NETWORK
TITLE =SK_A5_START_Molch_L  Anlage 5 Lampe Start Molch IM SIRUPRAUM
// Act 009
// Box           : AB-SK
// Output address: Q181.5
      CALL FC    70 (
           UnitNo                   := #UnitNo,
           ActRec                   := DB5050.SK_A5_START_Molch_L,
           Typ                      := 0,
           FBa                      := #xTmp,
           FBa2                     := #xTmp,
           Out                      := Q    181.5);

NETWORK
TITLE =SK_A5_MOLCH_BEI_A5_L  Anlage 5 Lampe Molch an A5 IM SIRUPRAUM
// Act 010
// Box           : AB-SK
// Output address: Q181.2
      CALL FC    70 (
           UnitNo                   := #UnitNo,
           ActRec                   := DB5050.SK_A5_MOLCH_BEI_A5_L,
           Typ                      := 0,
           FBa                      := #xTmp,
           FBa2                     := #xTmp,
           Out                      := Q    181.2);

NETWORK
TITLE =SK_A5_MOLCH_IN_SK_L  Anlage 5 Lampe Molch im SK IM SIRUPRAUM
// Act 011
// Box           : AB-SK
// Output address: Q181.3
      CALL FC    70 (
           UnitNo                   := #UnitNo,
           ActRec                   := DB5050.SK_A5_MOLCH_IN_SK_L,
           Typ                      := 0,
           FBa                      := #xTmp,
           FBa2                     := #xTmp,
           Out                      := Q    181.3);

NETWORK
TITLE =EA5_V1  MOLCH A5 V1
// Act 012
// Box           : VSA5
// Input address : I192.4
// Output address: Q192.4
      CALL FC    70 (
           UnitNo                   := #UnitNo,
           ActRec                   := DB5050.EA5_V1,
           Typ                      := 1,
           FBa                      := #xTmp,
           FBa2                     := I    192.4,
           Out                      := Q    192.4);

NETWORK
TITLE =EA5_V2  MOLCH A5 V2
// Act 013
// Box           : VSA5
// Input address : I192.5
// Output address: Q192.5
      CALL FC    70 (
           UnitNo                   := #UnitNo,
           ActRec                   := DB5050.EA5_V2,
           Typ                      := 1,
           FBa                      := #xTmp,
           FBa2                     := I    192.5,
           Out                      := Q    192.5);

NETWORK
TITLE =EA5_V31  MOLCH A5 V31 ohne RM
// Act 014
// Box           : VSA5
// Output address: Q192.0
      CALL FC    70 (
           UnitNo                   := #UnitNo,
           ActRec                   := DB5050.EA5_V31,
           Typ                      := 0,
           FBa                      := #xTmp,
           FBa2                     := #xTmp,
           Out                      := Q    192.0);

NETWORK
TITLE =EA5_V32  MOLCH A5 V31 ohne RM
// Act 015
// Box           : VSA5
// Input address : I192.1
// Output address: Q192.1
      CALL FC    70 (
           UnitNo                   := #UnitNo,
           ActRec                   := DB5050.EA5_V32,
           Typ                      := 0,
           FBa                      := #xTmp,
           FBa2                     := I    192.1,
           Out                      := Q    192.1);

NETWORK
TITLE =EA5_V41  MOLCH A5 V41
// Act 016
// Box           : VSA5
// Input address : I192.2
// Output address: Q192.2
      CALL FC    70 (
           UnitNo                   := #UnitNo,
           ActRec                   := DB5050.EA5_V41,
           Typ                      := 1,
           FBa                      := #xTmp,
           FBa2                     := I    192.2,
           Out                      := Q    192.2);

NETWORK
TITLE =EA5_V42  MOLCH A5 V42
// Act 017
// Box           : VSA5
// Input address : I192.3
// Output address: Q192.3
      CALL FC    70 (
           UnitNo                   := #UnitNo,
           ActRec                   := DB5050.EA5_V42,
           Typ                      := 1,
           FBa                      := #xTmp,
           FBa2                     := I    192.3,
           Out                      := Q    192.3);

NETWORK
TITLE =A5_MOLCH_LDT_Start  MOLCH A5 Reserve 23
// Act 019
// Box           : VSA5
// Output address: Q194.7
      CALL FC    70 (
           UnitNo                   := #UnitNo,
           ActRec                   := DB5050.A5_MOLCH_LDT_Start,
           Typ                      := 0,
           FBa                      := #xTmp,
           FBa2                     := #xTmp,
           Out                      := Q    194.7);

NETWORK
TITLE =Molch ist unterwegs(Mixer)


      CALL FC    70 (
           UnitNo                   := #UnitNo,
           ActRec                   := DB5050.Act20,
           Typ                      := 0,
           FBa                      := #xTmp,
           FBa2                     := #xTmp,
           Out                      := Q    199.3);

NETWORK
TITLE =Molch in Endposition (Mixer)


      CALL FC    70 (
           UnitNo                   := #UnitNo,
           ActRec                   := DB5050.Act21,
           Typ                      := 0,
           FBa                      := #xTmp,
           FBa2                     := #xTmp,
           Out                      := Q    199.7);

NETWORK
TITLE =A5_GOA501  Mixer A5 GOA501 Paneel CIP
// Act 025
// Box           : Mixer5
// Output address: Q199.2
      CALL FC    70 (
           UnitNo                   := #UnitNo,
           ActRec                   := DB5050.A5_GOA501,
           Typ                      := 0,
           FBa                      := #xTmp,
           FBa2                     := #xTmp,
           Out                      := Q    199.2);

NETWORK
TITLE =A5_GOA502  Mixer A5 GOA502 Paneel CIP
// Act 027
// Box           : Mixer5
// Output address: Q199.4
      CALL FC    70 (
           UnitNo                   := #UnitNo,
           ActRec                   := DB5050.A5_GOA502,
           Typ                      := 0,
           FBa                      := #xTmp,
           FBa2                     := #xTmp,
           Out                      := Q    199.4);

NETWORK
TITLE =A5_Schwenkbogen  "1"=CIP  "0"=Produktion
// Act 028
// Box           : Sirup
// Output address: DB_SEND_DOEHLER.Anlage5.Schwenkbogen
      CALL FC    70 (
           UnitNo                   := #UnitNo,
           ActRec                   := DB5050.A5_Schwenkbogen,
           Typ                      := 0,
           FBa                      := #xTmp,
           FBa2                     := #xTmp,
           Out                      := DB404.DBX   49.0);

NETWORK
TITLE =A5_GOA503  Mixer A5 GOA503 Paneel CIP
// Act 029
// Box           : Mixer5
// Output address: Q199.5
      CALL FC    70 (
           UnitNo                   := #UnitNo,
           ActRec                   := DB5050.A5_GOA503,
           Typ                      := 0,
           FBa                      := #xTmp,
           FBa2                     := #xTmp,
           Out                      := Q    199.5);

NETWORK
TITLE =VNI_A5_SCHWENKBOGEN_RL  Schwenkbogen A5-RL liegt richtig
// Act 042
// Box           : AB-SK
// Output address: Q183.1
      CALL FC    70 (
           UnitNo                   := #UnitNo,
           ActRec                   := DB5050.VNI_A5_SCHWENKBOGEN_RL,
           Typ                      := 0,
           FBa                      := #xTmp,
           FBa2                     := #xTmp,
           Out                      := Q    183.1);

NETWORK
TITLE =VNI_MOLCH_verr_A5  SIGNAL AN VNI Molch verriegelt an Anlage5
// Act 043
// Box           : AB-SK
// Output address: Q183.2
      CALL FC    70 (
           UnitNo                   := #UnitNo,
           ActRec                   := DB5050.VNI_MOLCH_verr_A5,
           Typ                      := 0,
           FBa                      := #xTmp,
           FBa2                     := #xTmp,
           Out                      := Q    183.2);

NETWORK
TITLE =VNI_MOLCH_Sender_A5  SIGNAL AN VNI Molch an Sendestation A5 (SK)
// Act 044
// Box           : AB-SK
// Output address: Q183.3
      CALL FC    70 (
           UnitNo                   := #UnitNo,
           ActRec                   := DB5050.VNI_MOLCH_Sender_A5,
           Typ                      := 0,
           FBa                      := #xTmp,
           FBa2                     := #xTmp,
           Out                      := Q    183.3);

NETWORK
TITLE =VNI_MOLCH_Empfang_A5  Molch an Empfangsstation (M5)
// Act 045
// Box           : AB-SK
// Output address: Q183.4
      CALL FC    70 (
           UnitNo                   := #UnitNo,
           ActRec                   := DB5050.VNI_MOLCH_Empfang_A5,
           Typ                      := 0,
           FBa                      := #xTmp,
           FBa2                     := #xTmp,
           Out                      := Q    183.4);

NETWORK
TITLE =A5_Molch_Sirup  "1"=Molch ist im Sirupraum
// Act 046
// Box           : Sirup
// Output address: DB_SEND_DOEHLER.Anlage5.Molch_Sirup
      CALL FC    70 (
           UnitNo                   := #UnitNo,
           ActRec                   := DB5050.A5_Molch_Sirup,
           Typ                      := 0,
           FBa                      := #xTmp,
           FBa2                     := #xTmp,
           Out                      := DB404.DBX   48.0);

NETWORK
TITLE =A5_Molch_Anlage  "1"=Molch ist an der Anlage
// Act 047
// Box           : Sirup
// Output address: DB_SEND_DOEHLER.Anlage5.Molch_Anlage
      CALL FC    70 (
           UnitNo                   := #UnitNo,
           ActRec                   := DB5050.A5_Molch_Anlage,
           Typ                      := 0,
           FBa                      := #xTmp,
           FBa2                     := #xTmp,
           Out                      := DB404.DBX   48.1);

NETWORK
TITLE =A5_Molch_PRO  "1"=Molch ist bereit für Produktion
// Act 048
// Box           : Sirup
// Output address: DB_SEND_DOEHLER.Anlage5.Molch_PRO
      CALL FC    70 (
           UnitNo                   := #UnitNo,
           ActRec                   := DB5050.A5_Molch_PRO,
           Typ                      := 0,
           FBa                      := #xTmp,
           FBa2                     := #xTmp,
           Out                      := DB404.DBX   48.2);

NETWORK
TITLE =A5_Molch_CIP  "1"=Molch ist bereit für CIP
// Act 049
// Box           : Sirup
// Output address: DB_SEND_DOEHLER.Anlage5.Molch_CIP
      CALL FC    70 (
           UnitNo                   := #UnitNo,
           ActRec                   := DB5050.A5_Molch_CIP,
           Typ                      := 0,
           FBa                      := #xTmp,
           FBa2                     := #xTmp,
           Out                      := DB404.DBX   48.3);

NETWORK
TITLE =A5_Sirupanforderung
// Act 050
// Box           : Sirup
// Output address: DB_SEND_DOEHLER.Anlage5.Sirupanforderung
      CALL FC    70 (
           UnitNo                   := #UnitNo,
           ActRec                   := DB5050.A5_Sirupanforderung,
           Typ                      := 0,
           FBa                      := #xTmp,
           FBa2                     := #xTmp,
           Out                      := DB404.DBX   48.4);

END_FUNCTION_BLOCK

FUNCTION_BLOCK FB 4051
TITLE =U105: Transfer Plant 5
FAMILY : BOTEC_F1
NAME : UniE
VERSION : 1.2


VAR_TEMP
  CIP : BOOL ;	//CIP active
  UNIM : BOOL ;	//Unit Not In Maintenance
  GenRel : BOOL ;	//general OK (emergency and maintenance OK)
  EStopOK : BOOL ;	//emergency OK
  UnitNo : INT ;	//unit number
  xTmp : BOOL ;	//Temporary Bool
  iTmp : INT ;	//Temporary INT
  rTmp : REAL ;	//Temporary REAL
  dTmp : DINT ;	//Temporary DINT (free for general use)
  RetValInt : INT ;	//return value
END_VAR
BEGIN
NETWORK
TITLE =General

      SET   ;
// Simulation ---------------------------------------------------------------
      A     DB4051.DBX 1357.7;
      CC    FB  4059; // "U105Sim"
      A     DB4051.DBX   17.3;
      =     DB4051.DBX 1357.7; //Help bit for simulation

// get unit number ----------------------------------------------------------
      L     DB4050.DBW    0;
      T     #UnitNo;

// communication ------------------------------------------------------------
      UC    FB  4055; // U105Com

NETWORK
TITLE =Sequence organisation

      CLR   ;
      =     M    122.2;

// sequencer ----------------------------------------------------------------
      A     DB4053.DBX   43.1;
      S     DB4053.DBX   97.3;

      CALL FC    40 (
           UnitNo                   := #UnitNo);

END_FUNCTION_BLOCK

FUNCTION_BLOCK FB 4070
TITLE =U107: Sirup Anlage  7
FAMILY : BOTEC_F1
NAME : U107A
VERSION : 2.1


VAR_TEMP
  EStopOK : BOOL ;	//auxiliary flag
  CIP : BOOL ;	//CIP Program Selected
  xTmp : BOOL ;	//Temporary Bool(free for general use)
  DummyBool : BOOL ;	//Temporary Bool(free for general use)
  UnitNo : INT ;	//unit number
  UnitFB : INT ;	//unit expansion FB number
  rTmp : REAL ;	//Temporary REAL (free for general use)
  iTmp : INT ;	//Temporary INT (free for general use)
  DummyInt : INT ;	//Temporary INT (free for general use)
  dTmp : DINT ;	//Temporary DINT (free for general use)
END_VAR
BEGIN
NETWORK
TITLE =general

      CLR   ;
      =     #xTmp;
      =     #EStopOK;

      L     DB4070.DBW    0;
      T     #UnitNo;
      L     DB4070.DBW    2;
      T     #UnitFB;

NETWORK
TITLE =Universal value

      NOP   0;
// unv001 UnV 001 Process Status
      CALL FC    27 (
           UnitNo                   := #UnitNo,
           UnVRec                   := DB5075.unv001,
           ValExt                   := DB5075.DBD  234);

// unv002 UnV 002 Universal Value 02
      CALL FC    27 (
           UnitNo                   := #UnitNo,
           UnVRec                   := DB5075.unv002,
           ValExt                   := DB5075.DBD  362);

// unv003 UnV 003 Universal Value 03
      CALL FC    27 (
           UnitNo                   := #UnitNo,
           UnVRec                   := DB5075.unv003,
           ValExt                   := DB5075.DBD  490);

// unv004 UnV 004 Universal Value 04
      CALL FC    27 (
           UnitNo                   := #UnitNo,
           UnVRec                   := DB5075.unv004,
           ValExt                   := DB5075.DBD  618);

NETWORK
TITLE =special inputs

      NOP   0;
// GOA_SA7_3_1_oben SpI 004
      CALL FC    14 (
           UnitNo                   := #UnitNo,
           SpIRec                   := DB5071.GOA_SA7_3_1_oben,
           SpIBit                   := I     74.2);

// GOA_SA7_3_2_unten SpI 005 Korb im Sirupraum in unterer Position
      CALL FC    14 (
           UnitNo                   := #UnitNo,
           SpIRec                   := DB5071.GOA_SA7_3_2_unten,
           SpIBit                   := I     74.3);

// GOA_SA7_1 SpI 006
      CALL FC    14 (
           UnitNo                   := #UnitNo,
           SpIRec                   := DB5071.GOA_SA7_1,
           SpIBit                   := I     74.1);// "GOA_SA7_1"

// GOA_SA7_2 SpI 007
      CALL FC    14 (
           UnitNo                   := #UnitNo,
           SpIRec                   := DB5071.GOA_SA7_2,
           SpIBit                   := I     74.0);//"GOA_SA7_2"

// SK_A7_Molch_Abbruch_DT SpI 008 MOLCH A7 Drucktaste Abbruch Sirupraum
      CALL FC    14 (
           UnitNo                   := #UnitNo,
           SpIRec                   := DB5071.SK_A7_Molch_Abbruch_DT,
           SpIBit                   := I    180.0);

// SK_A7_START_Molch_LDT SpI 009 MOLCH A7 L-Drucktaste Start Sirupraum
      CALL FC    14 (
           UnitNo                   := #UnitNo,
           SpIRec                   := DB5071.SK_A7_START_Molch_LDT,
           SpIBit                   := I    180.3);

// A7_Sk1_Handklappe SpI 010
      CALL FC    14 (
           UnitNo                   := #UnitNo,
           SpIRec                   := DB5071.A7_Sk1_Handklappe,
           SpIBit                   := I     74.7);

// GOA_EA7_3_1_oben SpI 014
      CALL FC    14 (
           UnitNo                   := #UnitNo,
           SpIRec                   := DB5071.GOA_EA7_3_1_oben,
           SpIBit                   := I     26.5);

// GOA_EA7_3_2_unten SpI 015
      CALL FC    14 (
           UnitNo                   := #UnitNo,
           SpIRec                   := DB5071.GOA_EA7_3_2_unten,
           SpIBit                   := I     26.6);

// GOA_EA7_3 SpI 016 Molch in Startposition an Anlage 7
      CALL FC    14 (
           UnitNo                   := #UnitNo,
           SpIRec                   := DB5071.GOA_EA7_3,
           SpIBit                   := I     26.3);

// GOA_EA7_4 SpI 017 GOA Molch in Ruhelage an Anlage 7
      CALL FC    14 (
           UnitNo                   := #UnitNo,
           SpIRec                   := DB5071.GOA_EA7_4,
           SpIBit                   := I     26.4);

// A7_SS_FRG_MOLCH SpI 018 Anlage 7 Schlüsselschalter Freigabe Molch
      CALL FC    14 (
           UnitNo                   := #UnitNo,
           SpIRec                   := DB5071.A7_SS_FRG_MOLCH,
           SpIBit                   := I     27.4);

// LDT_START_MOLCH_S2 SpI 019 STARTTASTER AB
      CALL FC    14 (
           UnitNo                   := #UnitNo,
           SpIRec                   := DB5071.LDT_START_MOLCH_S2,
           SpIBit                   := I     26.7);

// LDT_STOP_MOLCH_S2 SpI 020
      CALL FC    14 (
           UnitNo                   := #UnitNo,
           SpIRec                   := DB5071.LDT_STOP_MOLCH_S2,
           SpIBit                   := I     27.5);

// EA7_K2_Handklappe SpI 021 Handklappe Fueller 7
      CALL FC    14 (
           UnitNo                   := #UnitNo,
           SpIRec                   := DB5071.EA7_K2_Handklappe,
           SpIBit                   := I     27.2);

// GOA_701 SpI 022 Spare
      CALL FC    14 (
           UnitNo                   := #UnitNo,
           SpIRec                   := DB5071.GOA_701x,
           SpIBit                   := FALSE);

// GOA_702 SpI 023 Meldung an Fueller/Sirup Anl.7
      CALL FC    14 (
           UnitNo                   := #UnitNo,
           SpIRec                   := DB5071.GOA_702,
           SpIBit                   := I     26.1);

// GOA_701 SpI 025 Meldung an Fueller/Sirup Anl.7
      CALL FC    14 (
           UnitNo                   := #UnitNo,
           SpIRec                   := DB5071.GOA_701,
           SpIBit                   := I     26.0);

NETWORK
TITLE =messages

      NOP   0;
// msg001 Msg 001 Message 01
      CALL FC    16 (
           UnitNo                   := #UnitNo,
           MsgRec                   := DB5077.msg001,
           MsgBit                   := DB5077.DBX   82.7);

// msg002 Msg 002 Message 02
      CALL FC    16 (
           UnitNo                   := #UnitNo,
           MsgRec                   := DB5077.msg002,
           MsgBit                   := DB5077.DBX  142.7);

// msg003 Msg 003 Message 03
      CALL FC    16 (
           UnitNo                   := #UnitNo,
           MsgRec                   := DB5077.msg003,
           MsgBit                   := DB5077.DBX  202.7);

NETWORK
TITLE =unit supply

      UC    FB [#UnitFB];

NETWORK
TITLE =A7_MWV1  Ansteuerung A7_MWV1
// Act 002
// Box           : VSSK
// Input address : I72.4
// Output address: Q52.4
      CALL FC    70 (
           UnitNo                   := #UnitNo,
           ActRec                   := DB5070.A7_MWV1,
           Typ                      := 1,
           FBa                      := #xTmp,
           FBa2                     := I     72.4,
           Out                      := Q     52.4);

NETWORK
TITLE =SA7_V2  Ansteuerung SA7_V2
// Act 003
// Box           : VSSK
// Input address : I72.5
// Output address: Q52.5
      CALL FC    70 (
           UnitNo                   := #UnitNo,
           ActRec                   := DB5070.SA7_V2,
           Typ                      := 3,
           FBa                      := I     72.5,
           FBa2                     := #xTmp,
           Out                      := Q     52.5);

NETWORK
TITLE =SA7_V31  Ansteuerung SA7_V31 ohne RM
// Act 004
// Box           : VSSK
// Output address: Q52.0
      CALL FC    70 (
           UnitNo                   := #UnitNo,
           ActRec                   := DB5070.SA7_V31,
           Typ                      := 0,
           FBa                      := #xTmp,
           FBa2                     := #xTmp,
           Out                      := Q     52.0);

NETWORK
TITLE =SA7_V32  Ansteuerung SA7_V32 ohne RM
// Act 005
// Box           : VSSK
// Output address: Q52.1
      CALL FC    70 (
           UnitNo                   := #UnitNo,
           ActRec                   := DB5070.SA7_V32,
           Typ                      := 0,
           FBa                      := #xTmp,
           FBa2                     := #xTmp,
           Out                      := Q     52.1);

NETWORK
TITLE =SA7_V41  Ansteuerung SA7_V41
// Act 006
// Box           : VSSK
// Input address : I72.2
// Output address: Q52.2
      CALL FC    70 (
           UnitNo                   := #UnitNo,
           ActRec                   := DB5070.SA7_V41,
           Typ                      := 3,
           FBa                      := I     72.2,
           FBa2                     := #xTmp,
           Out                      := Q     52.2);

NETWORK
TITLE =SA7_V42  Ansteuerung SA7_V42
// Act 007
// Box           : VSSK
// Input address : I72.3
// Output address: Q52.3
      CALL FC    70 (
           UnitNo                   := #UnitNo,
           ActRec                   := DB5070.SA7_V42,
           Typ                      := 3,
           FBa                      := I     72.3,
           FBa2                     := #xTmp,
           Out                      := Q     52.3);

NETWORK
TITLE =SK_A7_Abbruch_L  Anlage 7 Lampe Abbruch IM SIRUPRAUM
// Act 008
// Box           : AB-SK
// Output address: Q180.2
      CALL FC    70 (
           UnitNo                   := #UnitNo,
           ActRec                   := DB5070.SK_A7_Abbruch_L,
           Typ                      := 0,
           FBa                      := #xTmp,
           FBa2                     := #xTmp,
           Out                      := Q    180.2);

NETWORK
TITLE =SK_A7_START_Molch_L  Anlage 7 Lampe Start Molch IM SIRUPRAUM
// Act 009
// Box           : AB-SK
// Output address: Q180.3
      CALL FC    70 (
           UnitNo                   := #UnitNo,
           ActRec                   := DB5070.SK_A7_START_Molch_L,
           Typ                      := 0,
           FBa                      := #xTmp,
           FBa2                     := #xTmp,
           Out                      := Q    180.3);

NETWORK
TITLE =SK_A7_MOLCH_BEI_A7_L  Anlage 7 Lampe Molch an A7 IM SIRUPRAUM
// Act 010
// Box           : AB-SK
// Output address: Q180.0
      CALL FC    70 (
           UnitNo                   := #UnitNo,
           ActRec                   := DB5070.SK_A7_MOLCH_BEI_A7_L,
           Typ                      := 0,
           FBa                      := #xTmp,
           FBa2                     := #xTmp,
           Out                      := Q    180.0);

NETWORK
TITLE =SK_A7_MOLCH_IN_SK_L  Anlage 7 Lampe Molch im SK IM SIRUPRAUM
// Act 011
// Box           : AB-SK
// Output address: Q180.1
      CALL FC    70 (
           UnitNo                   := #UnitNo,
           ActRec                   := DB5070.SK_A7_MOLCH_IN_SK_L,
           Typ                      := 0,
           FBa                      := #xTmp,
           FBa2                     := #xTmp,
           Out                      := Q    180.1);

NETWORK
TITLE =EA7_V1  Molch Anlage 7
// Act 012
// Box           : VSA7
// Input address : I24.4
// Output address: Q46.4
      CALL FC    70 (
           UnitNo                   := #UnitNo,
           ActRec                   := DB5070.EA7_V1,
           Typ                      := 3,
           FBa                      := I     24.4,
           FBa2                     := #xTmp,
           Out                      := Q     46.4);

NETWORK
TITLE =EA7_V2  Molch Anlage 7
// Act 013
// Box           : VSA7
// Input address : I24.5
// Output address: Q46.5
      CALL FC    70 (
           UnitNo                   := #UnitNo,
           ActRec                   := DB5070.EA7_V2,
           Typ                      := 3,
           FBa                      := I     24.5,
           FBa2                     := #xTmp,
           Out                      := Q     46.5);

NETWORK
TITLE =EA7_V31  Molch Anlage 7
// Act 014
// Box           : VSA7
// Output address: Q46.0
      CALL FC    70 (
           UnitNo                   := #UnitNo,
           ActRec                   := DB5070.EA7_V31,
           Typ                      := 0,
           FBa                      := #xTmp,
           FBa2                     := #xTmp,
           Out                      := Q     46.0);

NETWORK
TITLE =EA7_V32  Molch Anlage 7
// Act 015
// Box           : VSA7
// Output address: Q46.1
      CALL FC    70 (
           UnitNo                   := #UnitNo,
           ActRec                   := DB5070.EA7_V32,
           Typ                      := 0,
           FBa                      := #xTmp,
           FBa2                     := #xTmp,
           Out                      := Q     46.1);

NETWORK
TITLE =EA7_V41  Molch Anlage 7
// Act 016
// Box           : VSA7
// Input address : I24.2
// Output address: Q46.2
      CALL FC    70 (
           UnitNo                   := #UnitNo,
           ActRec                   := DB5070.EA7_V41,
           Typ                      := 3,
           FBa                      := I     24.2,
           FBa2                     := #xTmp,
           Out                      := Q     46.2);

NETWORK
TITLE =EA7_V42  Molch Anlage 7
// Act 017
// Box           : VSA7
// Input address : I24.3
// Output address: Q46.3
      CALL FC    70 (
           UnitNo                   := #UnitNo,
           ActRec                   := DB5070.EA7_V42,
           Typ                      := 3,
           FBa                      := I     24.3,
           FBa2                     := #xTmp,
           Out                      := Q     46.3);

NETWORK
TITLE =LA_S2_MOLCH_START  LAMPE LDT AB
// Act 019
// Box           : FRM-A7
// Output address: Q59.7
      CALL FC    70 (
           UnitNo                   := #UnitNo,
           ActRec                   := DB5070.LA_S2_MOLCH_START,
           Typ                      := 0,
           FBa                      := #xTmp,
           FBa2                     := #xTmp,
           Out                      := Q     59.7);

NETWORK
TITLE =Molch ist unterwegs (Mixer)


      CALL FC    70 (
           UnitNo                   := #UnitNo,
           ActRec                   := DB5070.Act20,
           Typ                      := 0,
           FBa                      := #xTmp,
           FBa2                     := #xTmp,
           Out                      := Q     59.3);

NETWORK
TITLE =Molch in Endposition (Mixer)


      CALL FC    70 (
           UnitNo                   := #UnitNo,
           ActRec                   := DB5070.Act21,
           Typ                      := 0,
           FBa                      := #xTmp,
           FBa2                     := #xTmp,
           Out                      := Q     59.6);

NETWORK
TITLE =A7_GOA_701  Meldung an Fueller/Sirup Anl.7
// Act 022
// Box           : FRM-A7
// Output address: Q59.2
      CALL FC    70 (
           UnitNo                   := #UnitNo,
           ActRec                   := DB5070.A7_GOA_701,
           Typ                      := 0,
           FBa                      := #xTmp,
           FBa2                     := #xTmp,
           Out                      := Q     59.2);

NETWORK
TITLE =A7_GOA_702  Meldung an Fueller/Mixer Anl.7
// Act 023
// Box           : FRM-A7
// Output address: Q59.5
      CALL FC    70 (
           UnitNo                   := #UnitNo,
           ActRec                   := DB5070.A7_GOA_702,
           Typ                      := 0,
           FBa                      := #xTmp,
           FBa2                     := #xTmp,
           Out                      := Q     59.5);

NETWORK
TITLE =A7_GOA_703  Meldung an Fueller/Mixer Anl.7
// Act 024
// Box           : FRM-A7
// Output address: Q59.4
      CALL FC    70 (
           UnitNo                   := #UnitNo,
           ActRec                   := DB5070.A7_GOA_703,
           Typ                      := 0,
           FBa                      := #xTmp,
           FBa2                     := #xTmp,
           Out                      := Q     59.4);

NETWORK
TITLE =A7_Schwenkbogen  "1"=CIP  "0"=Produktion
// Act 028
// Box           : Sirup
// Output address: DB_SEND_DOEHLER.Anlage7.Schwenkbogen
      CALL FC    70 (
           UnitNo                   := #UnitNo,
           ActRec                   := DB5070.A7_Schwenkbogen,
           Typ                      := 0,
           FBa                      := #xTmp,
           FBa2                     := #xTmp,
           Out                      := DB404.DBX   53.0);

NETWORK
TITLE =A7_Molch_Sirup  "1"=Molch ist im Sirupraum
// Act 046
// Box           : Sirup
// Output address: DB_SEND_DOEHLER.Anlage7.Molch_Sirup
      CALL FC    70 (
           UnitNo                   := #UnitNo,
           ActRec                   := DB5070.A7_Molch_Sirup,
           Typ                      := 0,
           FBa                      := #xTmp,
           FBa2                     := #xTmp,
           Out                      := DB404.DBX   52.0);

NETWORK
TITLE =A7_Molch_Anlage  "1"=Molch ist an der Anlage
// Act 047
// Box           : Sirup
// Output address: DB_SEND_DOEHLER.Anlage7.Molch_Anlage
      CALL FC    70 (
           UnitNo                   := #UnitNo,
           ActRec                   := DB5070.A7_Molch_Anlage,
           Typ                      := 0,
           FBa                      := #xTmp,
           FBa2                     := #xTmp,
           Out                      := DB404.DBX   52.1);

NETWORK
TITLE =A7_Molch_PRO  "1"=Molch ist bereit für Produktion
// Act 048
// Box           : Sirup
// Output address: DB_SEND_DOEHLER.Anlage7.Molch_PRO
      CALL FC    70 (
           UnitNo                   := #UnitNo,
           ActRec                   := DB5070.A7_Molch_PRO,
           Typ                      := 0,
           FBa                      := #xTmp,
           FBa2                     := #xTmp,
           Out                      := DB404.DBX   52.2);

NETWORK
TITLE =A7_Molch_CIP  "1"=Molch ist bereit für CIP
// Act 049
// Box           : Sirup
// Output address: DB_SEND_DOEHLER.Anlage7.Molch_CIP
      CALL FC    70 (
           UnitNo                   := #UnitNo,
           ActRec                   := DB5070.A7_Molch_CIP,
           Typ                      := 0,
           FBa                      := #xTmp,
           FBa2                     := #xTmp,
           Out                      := DB404.DBX   52.3);

NETWORK
TITLE =A7_Sirupanforderung
// Act 050
// Box           : Sirup
// Output address: DB_SEND_DOEHLER.Anlage7.Sirupanforderung
      CALL FC    70 (
           UnitNo                   := #UnitNo,
           ActRec                   := DB5070.A7_Sirupanforderung,
           Typ                      := 0,
           FBa                      := #xTmp,
           FBa2                     := #xTmp,
           Out                      := DB404.DBX   52.4);

END_FUNCTION_BLOCK

FUNCTION_BLOCK FB 4071
TITLE =U107: Transfer Plant 7
FAMILY : BOTEC_F1
NAME : UniE
VERSION : 1.2


VAR_TEMP
  CIP : BOOL ;	//CIP active
  UNIM : BOOL ;	//Unit Not In Maintenance
  GenRel : BOOL ;	//general OK (emergency and maintenance OK)
  EStopOK : BOOL ;	//emergency OK
  UnitNo : INT ;	//unit number
  xTmp : BOOL ;	//Temporary Bool
  iTmp : INT ;	//Temporary INT
  rTmp : REAL ;	//Temporary REAL
  dTmp : DINT ;	//Temporary DINT (free for general use)
  RetValInt : INT ;	//return value
END_VAR
BEGIN
NETWORK
TITLE =General

      SET   ;
// Simulation ---------------------------------------------------------------
      A     DB4071.DBX 1357.7;
      CC    FB  4079; // "U107Sim"
      A     DB4071.DBX   17.3;
      =     DB4071.DBX 1357.7; //Help bit for simulation

// get unit number ----------------------------------------------------------
      L     DB4070.DBW    0;
      T     #UnitNo;

// CIP ----------------------------------------------------------------------
      L     DB4071.DBD   54;
      L     0;
      <D    ;
      =     #CIP;

// emergency OK -------------------------------------------------------------
      A     DB4075.DBX   27.0; //Emergency Stop OK
      =     #EStopOK;

// Write Unit in Maintenance ------------------------------------------------

      AN    DB4071.DBX   69.7;
      =     #UNIM;

// emergency and maintenance OK ---------------------------------------------
      A     #EStopOK;
      A     #UNIM;
      =     #GenRel;

// communication ------------------------------------------------------------
      UC    FB  4075; // U107Com

NETWORK
TITLE =Sequence organisation

      CLR   ;
      =     M    122.2;

// SFM supply ----------------------------------------------------------------

// sequencer ----------------------------------------------------------------
      A     DB4073.DBX   43.1;
      S     DB4073.DBX   97.3;

      CALL FC    40 (
           UnitNo                   := #UnitNo);

END_FUNCTION_BLOCK

FUNCTION_BLOCK FB 4080
TITLE =U108: Sirup Anlage  8
FAMILY : BOTEC_F1
NAME : U108A
VERSION : 2.1


VAR_TEMP
  EStopOK : BOOL ;	//auxiliary flag
  CIP : BOOL ;	//CIP Program Selected
  xTmp : BOOL ;	//Temporary Bool(free for general use)
  DummyBool : BOOL ;	//Temporary Bool(free for general use)
  UnitNo : INT ;	//unit number
  UnitFB : INT ;	//unit expansion FB number
  rTmp : REAL ;	//Temporary REAL (free for general use)
  iTmp : INT ;	//Temporary INT (free for general use)
  DummyInt : INT ;	//Temporary INT (free for general use)
  dTmp : DINT ;	//Temporary DINT (free for general use)
END_VAR
BEGIN
NETWORK
TITLE =general

      CLR   ;
      =     #xTmp;
      =     #EStopOK;

      L     DB4080.DBW    0;
      T     #UnitNo;
      L     DB4080.DBW    2;
      T     #UnitFB;

NETWORK
TITLE =Universal value

      NOP   0;
// unv001 UnV 001 Process Status
      CALL FC    27 (
           UnitNo                   := #UnitNo,
           UnVRec                   := DB5085.unv001,
           ValExt                   := DB5085.DBD  234);

// unv002 UnV 002 Universal Value 02
      CALL FC    27 (
           UnitNo                   := #UnitNo,
           UnVRec                   := DB5085.unv002,
           ValExt                   := DB5085.DBD  362);

// unv003 UnV 003 Universal Value 03
      CALL FC    27 (
           UnitNo                   := #UnitNo,
           UnVRec                   := DB5085.unv003,
           ValExt                   := DB5085.DBD  490);

// unv004 UnV 004 Universal Value 04
      CALL FC    27 (
           UnitNo                   := #UnitNo,
           UnVRec                   := DB5085.unv004,
           ValExt                   := DB5085.DBD  618);

NETWORK
TITLE =messages

      NOP   0;
// msg001 Msg 001 Message 01
      CALL FC    16 (
           UnitNo                   := #UnitNo,
           MsgRec                   := DB5087.msg001,
           MsgBit                   := DB5087.DBX   82.7);

// msg002 Msg 002 Message 02
      CALL FC    16 (
           UnitNo                   := #UnitNo,
           MsgRec                   := DB5087.msg002,
           MsgBit                   := DB5087.DBX  142.7);

// msg003 Msg 003 Message 03
      CALL FC    16 (
           UnitNo                   := #UnitNo,
           MsgRec                   := DB5087.msg003,
           MsgBit                   := DB5087.DBX  202.7);

NETWORK
TITLE =unit supply

      UC    FB [#UnitFB];
END_FUNCTION_BLOCK

FUNCTION_BLOCK FB 4081
TITLE =U108: Transfer Plant 8
FAMILY : BOTEC_F1
NAME : UniE
VERSION : 1.2


VAR_TEMP
  CIP : BOOL ;	//CIP active
  UNIM : BOOL ;	//Unit Not In Maintenance
  GenRel : BOOL ;	//general OK (emergency and maintenance OK)
  EStopOK : BOOL ;	//emergency OK
  UnitNo : INT ;	//unit number
  xTmp : BOOL ;	//Temporary Bool
  iTmp : INT ;	//Temporary INT
  rTmp : REAL ;	//Temporary REAL
  dTmp : DINT ;	//Temporary DINT (free for general use)
  RetValInt : INT ;	//return value
END_VAR
BEGIN
NETWORK
TITLE =General

      SET   ;
// Simulation ---------------------------------------------------------------
      A     DB4081.DBX 1357.7;
      CC    FB  4089; // "U108Sim"
      A     DB4081.DBX   17.3;
      =     DB4081.DBX 1357.7; //Help bit for simulation

// get unit number ----------------------------------------------------------
      L     DB4080.DBW    0;
      T     #UnitNo;

// CIP ----------------------------------------------------------------------
      L     DB4081.DBD   54;
      L     0;
      <D    ;
      =     #CIP;

// emergency OK -------------------------------------------------------------
      A     DB4085.DBX   27.0; //Emergency Stop OK
      =     #EStopOK;

// Write Unit in Maintenance ------------------------------------------------

      AN    DB4081.DBX   69.7;
      =     #UNIM;

// emergency and maintenance OK ---------------------------------------------
      A     #EStopOK;
      A     #UNIM;
      =     #GenRel;

// communication ------------------------------------------------------------
      UC    FB  4085; // U108Com

NETWORK
TITLE =Universal Value

      NOP   0;

// ----------------------------------------------------------
// unv001 Process Status
// ----------------------------------------------------------
// process value to UnV
//      L     0.000000e+000
//      T     "U108UnVD".unv001.ValExt

// ----------------------------------------------------------
// unv002 Universal Value 02
// ----------------------------------------------------------
// process value to UnV
//      L     0.000000e+000
//      T     "U108UnVD".unv002.ValExt

// ----------------------------------------------------------
// unv003 Universal Value 03
// ----------------------------------------------------------
// process value to UnV
//      L     0.000000e+000
//      T     "U108UnVD".unv003.ValExt

// ----------------------------------------------------------
// unv004 Universal Value 04
// ----------------------------------------------------------
// process value to UnV
//      L     0.000000e+000
//      T     "U108UnVD".unv004.ValExt

NETWORK
TITLE =Messages

      NOP   0;

// ----------------------------------------------------------
// msg001 Message 01
// ----------------------------------------------------------
      SET   ;
      R     DB5087.DBX   80.7;
      =     DB5087.DBX   81.4;

      CLR   ;
      =     DB5087.DBX   82.7;

// ----------------------------------------------------------
// msg002 Message 02
// ----------------------------------------------------------
      SET   ;
      R     DB5087.DBX  140.7;
      =     DB5087.DBX  141.4;

      CLR   ;
      =     DB5087.DBX  142.7;

// ----------------------------------------------------------
// msg003 Message 03
// ----------------------------------------------------------
      SET   ;
      R     DB5087.DBX  200.7;
      =     DB5087.DBX  201.4;

      CLR   ;
      =     DB5087.DBX  202.7;

NETWORK
TITLE =Sequence organisation

      CLR   ;
      =     M    122.2;

// SFM supply ----------------------------------------------------------------

// sequencer ----------------------------------------------------------------
      A     DB4083.DBX   43.1;
      S     DB4083.DBX   97.3;

      CALL FC    40 (
           UnitNo                   := #UnitNo);

NETWORK
TITLE =Auto / Manual

      SET   ;
      AN    M    122.2;
      JC    MODE;
      AN    M    120.1;




MODE: SET   ;

END_FUNCTION_BLOCK

FUNCTION_BLOCK FB 4090
TITLE =U109: Sirup Anlage  9
FAMILY : BOTEC_F1
NAME : U109A
VERSION : 2.1


VAR_TEMP
  EStopOK : BOOL ;	//auxiliary flag
  CIP : BOOL ;	//CIP Program Selected
  xTmp : BOOL ;	//Temporary Bool(free for general use)
  DummyBool : BOOL ;	//Temporary Bool(free for general use)
  UnitNo : INT ;	//unit number
  UnitFB : INT ;	//unit expansion FB number
  rTmp : REAL ;	//Temporary REAL (free for general use)
  iTmp : INT ;	//Temporary INT (free for general use)
  DummyInt : INT ;	//Temporary INT (free for general use)
  dTmp : DINT ;	//Temporary DINT (free for general use)
END_VAR
BEGIN
NETWORK
TITLE =general

      CLR   ;
      =     #xTmp;
      =     #EStopOK;

      L     DB4090.DBW    0;
      T     #UnitNo;
      L     DB4090.DBW    2;
      T     #UnitFB;

NETWORK
TITLE =Universal value

      NOP   0;
// unv001 UnV 001 Process Status
      CALL FC    27 (
           UnitNo                   := #UnitNo,
           UnVRec                   := DB5095.unv001,
           ValExt                   := DB5095.DBD  234);

// unv002 UnV 002 Universal Value 02
      CALL FC    27 (
           UnitNo                   := #UnitNo,
           UnVRec                   := DB5095.unv002,
           ValExt                   := DB5095.DBD  362);

// unv003 UnV 003 Universal Value 03
      CALL FC    27 (
           UnitNo                   := #UnitNo,
           UnVRec                   := DB5095.unv003,
           ValExt                   := DB5095.DBD  490);

// unv004 UnV 004 Universal Value 04
      CALL FC    27 (
           UnitNo                   := #UnitNo,
           UnVRec                   := DB5095.unv004,
           ValExt                   := DB5095.DBD  618);

NETWORK
TITLE =special inputs

      NOP   0;
// GOA_SA9_31_oben SpI 004
      CALL FC    14 (
           UnitNo                   := #UnitNo,
           SpIRec                   := DB5091.GOA_SA9_31_oben,
           SpIBit                   := I     75.0);

// GOA_SA9_32_unten SpI 005 Korb im Sirupraum in unterer Position
      CALL FC    14 (
           UnitNo                   := #UnitNo,
           SpIRec                   := DB5091.GOA_SA9_32_unten,
           SpIBit                   := I     75.1);

// GOA_SA9_1 SpI 006
      CALL FC    14 (
           UnitNo                   := #UnitNo,
           SpIRec                   := DB5091.GOA_SA9_1,
           SpIBit                   := I     74.5);

// GOA_SA9_2 SpI 007
      CALL FC    14 (
           UnitNo                   := #UnitNo,
           SpIRec                   := DB5091.GOA_SA9_2,
           SpIBit                   := I     74.6);

// SK_A9_Molch_Abbruch_DT SpI 008 MOLCH A9 Drucktaste Abbruch Sirupraum
      CALL FC    14 (
           UnitNo                   := #UnitNo,
           SpIRec                   := DB5091.SK_A9_Molch_Abbruch_DT,
           SpIBit                   := I    180.5);

// SK_A9_START_Molch_LDT SpI 009 MOLCH A9 L-Drucktaste Start Sirupraum
      CALL FC    14 (
           UnitNo                   := #UnitNo,
           SpIRec                   := DB5091.SK_A9_START_Molch_LDT,
           SpIBit                   := I    181.0);

// A9_Sk1_Handklappe SpI 010
      CALL FC    14 (
           UnitNo                   := #UnitNo,
           SpIRec                   := DB5091.A9_Sk1_Handklappe,
           SpIBit                   := I     75.2);

// GOA_EA9_31_oben SpI 014 geändert 07.11.01
      CALL FC    14 (
           UnitNo                   := #UnitNo,
           SpIRec                   := DB5091.GOA_EA9_31_oben,
           SpIBit                   := I    176.5);

// GOA_EA9_32_unten SpI 015 geändert 07.11.01
      CALL FC    14 (
           UnitNo                   := #UnitNo,
           SpIRec                   := DB5091.GOA_EA9_32_unten,
           SpIBit                   := I    176.6);

// GOA_EA9_3 SpI 016 geändert 07.11.01
      CALL FC    14 (
           UnitNo                   := #UnitNo,
           SpIRec                   := DB5091.GOA_EA9_3,
           SpIBit                   := I    176.3);

// GOA_EA9_4 SpI 017 geändert 07.11.01
      CALL FC    14 (
           UnitNo                   := #UnitNo,
           SpIRec                   := DB5091.GOA_EA9_4,
           SpIBit                   := I    176.4);

// A9_SS_FRG_MOLCH SpI 018 Anlage 9 Schlüsselschalter Freigabe Molch
      CALL FC    14 (
           UnitNo                   := #UnitNo,
           SpIRec                   := DB5091.A9_SS_FRG_MOLCH,
           SpIBit                   := I    177.4);

// A9_Molch_LDT_Start SpI 019 geändert 07.11.01
      CALL FC    14 (
           UnitNo                   := #UnitNo,
           SpIRec                   := DB5091.A9_Molch_LDT_Start,
           SpIBit                   := I    176.7);

// A9_Molch_LDT_Stop SpI 020
      CALL FC    14 (
           UnitNo                   := #UnitNo,
           SpIRec                   := DB5091.A9_Molch_LDT_Stop,
           SpIBit                   := I    177.5);

// A9_K2_Handklappe SpI 021 geändert 07.11.01
      CALL FC    14 (
           UnitNo                   := #UnitNo,
           SpIRec                   := DB5091.A9_K2_Handklappe,
           SpIBit                   := I    177.2);

// GOA_901 SpI 022 geändert 07.11.01
      CALL FC    14 (
           UnitNo                   := #UnitNo,
           SpIRec                   := DB5091.GOA_901,
           SpIBit                   := I    176.0);

// GOA_902 SpI 023 geändert 07.11.01
      CALL FC    14 (
           UnitNo                   := #UnitNo,
           SpIRec                   := DB5091.GOA_902,
           SpIBit                   := I    176.1);

// EA9_K1_Handklappe SpI 024 Handklappe Fueller 9
      CALL FC    14 (
           UnitNo                   := #UnitNo,
           SpIRec                   := DB5091.EA9_K1_Handklappe,
           SpIBit                   := I    177.7);

// GOA_904 SpI 025
      CALL FC    14 (
           UnitNo                   := #UnitNo,
           SpIRec                   := DB5091.GOA_904,
           SpIBit                   := I    177.1);

NETWORK
TITLE =messages

      NOP   0;
// msg001 Msg 001 Message 01
      CALL FC    16 (
           UnitNo                   := #UnitNo,
           MsgRec                   := DB5097.msg001,
           MsgBit                   := DB5097.DBX   82.7);

// msg002 Msg 002 Message 02
      CALL FC    16 (
           UnitNo                   := #UnitNo,
           MsgRec                   := DB5097.msg002,
           MsgBit                   := DB5097.DBX  142.7);

// msg003 Msg 003 Message 03
      CALL FC    16 (
           UnitNo                   := #UnitNo,
           MsgRec                   := DB5097.msg003,
           MsgBit                   := DB5097.DBX  202.7);

NETWORK
TITLE =unit supply

      UC    FB [#UnitFB];

NETWORK
TITLE =A9_MWV1  Ansteuerung A9_MWV1
// Act 002
// Box           : VSSK
// Input address : I73.2
// Output address: Q53.2
      CALL FC    70 (
           UnitNo                   := #UnitNo,
           ActRec                   := DB5090.A9_MWV1,
           Typ                      := 1,
           FBa                      := #xTmp,
           FBa2                     := I     73.2,
           Out                      := Q     53.2);

NETWORK
TITLE =SA9_V2  Ansteuerung SA9_V2
// Act 003
// Box           : VSSK
// Input address : I73.3
// Output address: Q53.3
      CALL FC    70 (
           UnitNo                   := #UnitNo,
           ActRec                   := DB5090.SA9_V2,
           Typ                      := 1,
           FBa                      := #xTmp,
           FBa2                     := I     73.3,
           Out                      := Q     53.3);

NETWORK
TITLE =SA9_V31  Ansteuerung SA9_V31 ohne RM
// Act 004
// Box           : VSSK
// Output address: Q52.6
      CALL FC    70 (
           UnitNo                   := #UnitNo,
           ActRec                   := DB5090.SA9_V31,
           Typ                      := 0,
           FBa                      := #xTmp,
           FBa2                     := #xTmp,
           Out                      := Q     52.6);

NETWORK
TITLE =SA9_V32  Ansteuerung SA9_V32 ohne RM
// Act 005
// Box           : VSSK
// Output address: Q52.7
      CALL FC    70 (
           UnitNo                   := #UnitNo,
           ActRec                   := DB5090.SA9_V32,
           Typ                      := 0,
           FBa                      := #xTmp,
           FBa2                     := #xTmp,
           Out                      := Q     52.7);

NETWORK
TITLE =SA9_V41  Ansteuerung SA9_V41
// Act 006
// Box           : VSSK
// Input address : I73.0
// Output address: Q53.0
      CALL FC    70 (
           UnitNo                   := #UnitNo,
           ActRec                   := DB5090.SA9_V41,
           Typ                      := 1,
           FBa                      := #xTmp,
           FBa2                     := I     73.0,
           Out                      := Q     53.0);

NETWORK
TITLE =SA9_V42  Ansteuerung SA9_V42
// Act 007
// Box           : VSSK
// Input address : I73.1
// Output address: Q53.1
      CALL FC    70 (
           UnitNo                   := #UnitNo,
           ActRec                   := DB5090.SA9_V42,
           Typ                      := 1,
           FBa                      := #xTmp,
           FBa2                     := I     73.1,
           Out                      := Q     53.1);

NETWORK
TITLE =SK_A9_Abbruch_L  Anlage 9 Lampe Abbruch IM SIRUPRAUM
// Act 008
// Box           : AB-SK
// Output address: Q180.7
      CALL FC    70 (
           UnitNo                   := #UnitNo,
           ActRec                   := DB5090.SK_A9_Abbruch_L,
           Typ                      := 0,
           FBa                      := #xTmp,
           FBa2                     := #xTmp,
           Out                      := Q    180.7);

NETWORK
TITLE =SK_A9_START_Molch_L  Anlage 9 Lampe Start Molch IM SIRUPRAUM
// Act 009
// Box           : AB-SK
// Output address: Q181.0
      CALL FC    70 (
           UnitNo                   := #UnitNo,
           ActRec                   := DB5090.SK_A9_START_Molch_L,
           Typ                      := 0,
           FBa                      := #xTmp,
           FBa2                     := #xTmp,
           Out                      := Q    181.0);

NETWORK
TITLE =SK_A9_MOLCH_BEI_A9_L  Anlage 9 Lampe Molch an A11 IM SIRUPRAUM
// Act 010
// Box           : AB-SK
// Output address: Q180.5
      CALL FC    70 (
           UnitNo                   := #UnitNo,
           ActRec                   := DB5090.SK_A9_MOLCH_BEI_A9_L,
           Typ                      := 0,
           FBa                      := #xTmp,
           FBa2                     := #xTmp,
           Out                      := Q    180.5);

NETWORK
TITLE =SK_A9_MOLCH_IN_SK_L  Anlage 9 Lampe Molch im SK IM SIRUPRAUM
// Act 011
// Box           : AB-SK
// Output address: Q180.6
      CALL FC    70 (
           UnitNo                   := #UnitNo,
           ActRec                   := DB5090.SK_A9_MOLCH_IN_SK_L,
           Typ                      := 0,
           FBa                      := #xTmp,
           FBa2                     := #xTmp,
           Out                      := Q    180.6);

NETWORK
TITLE =EA9_V1  A9 V1
// Act 012
// Box           : VSA11
// Input address : I174.4
// Output address: Q174.4
      CALL FC    70 (
           UnitNo                   := #UnitNo,
           ActRec                   := DB5090.EA9_V1,
           Typ                      := 1,
           FBa                      := #xTmp,
           FBa2                     := I    174.4,
           Out                      := Q    174.4);

NETWORK
TITLE =EA9_V2  A9 V2
// Act 013
// Box           : VSA11
// Input address : I174.5
// Output address: Q174.5
      CALL FC    70 (
           UnitNo                   := #UnitNo,
           ActRec                   := DB5090.EA9_V2,
           Typ                      := 1,
           FBa                      := #xTmp,
           FBa2                     := I    174.5,
           Out                      := Q    174.5);

NETWORK
TITLE =EA9_V31  A9 V31 ohne RM
// Act 014
// Box           : VSA11
// Output address: Q174.0
      CALL FC    70 (
           UnitNo                   := #UnitNo,
           ActRec                   := DB5090.EA9_V31,
           Typ                      := 0,
           FBa                      := #xTmp,
           FBa2                     := #xTmp,
           Out                      := Q    174.0);

NETWORK
TITLE =EA9_V32  A9 V31 ohne RM
// Act 015
// Box           : VSA11
// Output address: Q174.1
      CALL FC    70 (
           UnitNo                   := #UnitNo,
           ActRec                   := DB5090.EA9_V32,
           Typ                      := 0,
           FBa                      := #xTmp,
           FBa2                     := #xTmp,
           Out                      := Q    174.1);

NETWORK
TITLE =EA9_V41  A9 V41
// Act 016
// Box           : VSA11
// Input address : I174.2
// Output address: Q174.2
      CALL FC    70 (
           UnitNo                   := #UnitNo,
           ActRec                   := DB5090.EA9_V41,
           Typ                      := 1,
           FBa                      := #xTmp,
           FBa2                     := I    174.2,
           Out                      := Q    174.2);

NETWORK
TITLE =EA9_V42  A9 V42
// Act 017
// Box           : VSA11
// Input address : I174.3
// Output address: Q174.3
      CALL FC    70 (
           UnitNo                   := #UnitNo,
           ActRec                   := DB5090.EA9_V42,
           Typ                      := 1,
           FBa                      := #xTmp,
           FBa2                     := I    174.3,
           Out                      := Q    174.3);

NETWORK
TITLE =EA9_MOLCH_LDT_Start  Lampe Start Molchen an Anlage 9
// Act 019
// Box           : VSA11
// Output address: Q176.7
      CALL FC    70 (
           UnitNo                   := #UnitNo,
           ActRec                   := DB5090.EA9_MOLCH_LDT_Start,
           Typ                      := 0,
           FBa                      := #xTmp,
           FBa2                     := #xTmp,
           Out                      := Q    176.7);

NETWORK
TITLE =Molch ist unterwegs (Mixer)


      CALL FC    70 (
           UnitNo                   := #UnitNo,
           ActRec                   := DB5090.Act20,
           Typ                      := 0,
           FBa                      := #xTmp,
           FBa2                     := #xTmp,
           Out                      := Q    171.3);

NETWORK
TITLE =Molch in Endposition (Mixer)


      CALL FC    70 (
           UnitNo                   := #UnitNo,
           ActRec                   := DB5090.Act21,
           Typ                      := 0,
           FBa                      := #xTmp,
           FBa2                     := #xTmp,
           Out                      := Q    171.7);

NETWORK
TITLE =A9_Schwenkbogen  "1"=CIP  "0"=Produktion
// Act 028
// Box           : Sirup
// Output address: DB_SEND_DOEHLER.Anlage9.Schwenkbogen
      CALL FC    70 (
           UnitNo                   := #UnitNo,
           ActRec                   := DB5090.A9_Schwenkbogen,
           Typ                      := 0,
           FBa                      := #xTmp,
           FBa2                     := #xTmp,
           Out                      := DB404.DBX   57.0);

NETWORK
TITLE =A9_Molch_Sirup  "1"=Molch ist im Sirupraum
// Act 046
// Box           : Sirup
// Output address: DB_SEND_DOEHLER.Anlage9.Molch_Sirup
      CALL FC    70 (
           UnitNo                   := #UnitNo,
           ActRec                   := DB5090.A9_Molch_Sirup,
           Typ                      := 0,
           FBa                      := #xTmp,
           FBa2                     := #xTmp,
           Out                      := DB404.DBX   56.0);

NETWORK
TITLE =A9_Molch_Anlage  "1"=Molch ist an der Anlage
// Act 047
// Box           : Sirup
// Output address: DB_SEND_DOEHLER.Anlage9.Molch_Anlage
      CALL FC    70 (
           UnitNo                   := #UnitNo,
           ActRec                   := DB5090.A9_Molch_Anlage,
           Typ                      := 0,
           FBa                      := #xTmp,
           FBa2                     := #xTmp,
           Out                      := DB404.DBX   56.1);

NETWORK
TITLE =A9_Molch_PRO  "1"=Molch ist bereit für Produktion
// Act 048
// Box           : Sirup
// Output address: DB_SEND_DOEHLER.Anlage9.Molch_PRO
      CALL FC    70 (
           UnitNo                   := #UnitNo,
           ActRec                   := DB5090.A9_Molch_PRO,
           Typ                      := 0,
           FBa                      := #xTmp,
           FBa2                     := #xTmp,
           Out                      := DB404.DBX   56.2);

NETWORK
TITLE =A9_Molch_CIP  "1"=Molch ist bereit für CIP
// Act 049
// Box           : Sirup
// Output address: DB_SEND_DOEHLER.Anlage9.Molch_CIP
      CALL FC    70 (
           UnitNo                   := #UnitNo,
           ActRec                   := DB5090.A9_Molch_CIP,
           Typ                      := 0,
           FBa                      := #xTmp,
           FBa2                     := #xTmp,
           Out                      := DB404.DBX   56.3);

NETWORK
TITLE =A9_Sirupanforderung
// Act 050
// Box           : Sirup
// Output address: DB_SEND_DOEHLER.Anlage9.Sirupanforderung
      CALL FC    70 (
           UnitNo                   := #UnitNo,
           ActRec                   := DB5090.A9_Sirupanforderung,
           Typ                      := 0,
           FBa                      := #xTmp,
           FBa2                     := #xTmp,
           Out                      := DB404.DBX   56.4);

END_FUNCTION_BLOCK

FUNCTION_BLOCK FB 4091
TITLE =U109: Transfer Plant 9
FAMILY : BOTEC_F1
NAME : UniE
VERSION : 1.2


VAR_TEMP
  CIP : BOOL ;	//CIP active
  UNIM : BOOL ;	//Unit Not In Maintenance
  GenRel : BOOL ;	//general OK (emergency and maintenance OK)
  EStopOK : BOOL ;	//emergency OK
  UnitNo : INT ;	//unit number
  xTmp : BOOL ;	//Temporary Bool
  iTmp : INT ;	//Temporary INT
  rTmp : REAL ;	//Temporary REAL
  dTmp : DINT ;	//Temporary DINT (free for general use)
  RetValInt : INT ;	//return value
END_VAR
BEGIN
NETWORK
TITLE =General

      SET   ;
// Simulation ---------------------------------------------------------------
      A     DB4091.DBX 1357.7;
      CC    FB  4099; // "U109Sim"
      A     DB4091.DBX   17.3;
      =     DB4091.DBX 1357.7; //Help bit for simulation

// get unit number ----------------------------------------------------------
      L     DB4090.DBW    0;
      T     #UnitNo;

// communication ------------------------------------------------------------
      UC    FB  4095; // U109Com

NETWORK
TITLE =Sequence organisation

      CLR   ;
      =     M    122.2;


// sequencer ----------------------------------------------------------------
      A     DB4093.DBX   43.1;
      S     DB4093.DBX   97.3;

      CALL FC    40 (
           UnitNo                   := #UnitNo);

END_FUNCTION_BLOCK

FUNCTION_BLOCK FB 4110
TITLE =U111: Sirup Anlage 11
FAMILY : BOTEC_F1
NAME : U111A
VERSION : 2.1


VAR_TEMP
  EStopOK : BOOL ;	//auxiliary flag
  CIP : BOOL ;	//CIP Program Selected
  xTmp : BOOL ;	//Temporary Bool(free for general use)
  DummyBool : BOOL ;	//Temporary Bool(free for general use)
  UnitNo : INT ;	//unit number
  UnitFB : INT ;	//unit expansion FB number
  rTmp : REAL ;	//Temporary REAL (free for general use)
  iTmp : INT ;	//Temporary INT (free for general use)
  DummyInt : INT ;	//Temporary INT (free for general use)
  dTmp : DINT ;	//Temporary DINT (free for general use)
END_VAR
BEGIN
NETWORK
TITLE =general

      BEU   ;

      CLR   ;
      =     #xTmp;
      =     #EStopOK;

      L     DB4110.DBW    0;
      T     #UnitNo;
      L     DB4110.DBW    2;
      T     #UnitFB;

NETWORK
TITLE =Universal value

      NOP   0;
// unv001 UnV 001 Process Status
      CALL FC    27 (
           UnitNo                   := #UnitNo,
           UnVRec                   := DB5115.unv001,
           ValExt                   := DB5115.DBD  234);

// unv002 UnV 002 Universal Value 02
      CALL FC    27 (
           UnitNo                   := #UnitNo,
           UnVRec                   := DB5115.unv002,
           ValExt                   := DB5115.DBD  362);

// unv003 UnV 003 Universal Value 03
      CALL FC    27 (
           UnitNo                   := #UnitNo,
           UnVRec                   := DB5115.unv003,
           ValExt                   := DB5115.DBD  490);

// unv004 UnV 004 Universal Value 04
      CALL FC    27 (
           UnitNo                   := #UnitNo,
           UnVRec                   := DB5115.unv004,
           ValExt                   := DB5115.DBD  618);

NETWORK
TITLE =special inputs

      NOP   0;
// U111_SpI034 SpI 034 spare
      CALL FC    14 (
           UnitNo                   := #UnitNo,
           SpIRec                   := DB5111.U111_SpI034,
           SpIBit                   := #DummyBool);

NETWORK
TITLE =messages

      NOP   0;
// msg001 Msg 001 Message 01
      CALL FC    16 (
           UnitNo                   := #UnitNo,
           MsgRec                   := DB5117.msg001,
           MsgBit                   := DB5117.DBX   82.7);

// msg002 Msg 002 Message 02
      CALL FC    16 (
           UnitNo                   := #UnitNo,
           MsgRec                   := DB5117.msg002,
           MsgBit                   := DB5117.DBX  142.7);

// msg003 Msg 003 Message 03
      CALL FC    16 (
           UnitNo                   := #UnitNo,
           MsgRec                   := DB5117.msg003,
           MsgBit                   := DB5117.DBX  202.7);

NETWORK
TITLE =unit supply

      UC    FB [#UnitFB];

NETWORK
TITLE =M11_K2_Handklappe  Mixer A11 Handklappe Sirupleitung
// Act 020
// Box           : FM-A11
// Output address: Q171.6
      CALL FC    70 (
           UnitNo                   := #UnitNo,
           ActRec                   := DB5110.M11_K2_Handklappe,
           Typ                      := 0,
           FBa                      := #xTmp,
           FBa2                     := #xTmp,
           Out                      := Q    171.6);

NETWORK
TITLE =A11_GOA_1101  Mixer A11 KEINE ANSTEUERUNG!!!
// Act 022
// Box           : FM-A11
// Output address: Q171.2
      CALL FC    70 (
           UnitNo                   := #UnitNo,
           ActRec                   := DB5110.A11_GOA_1101,
           Typ                      := 0,
           FBa                      := #xTmp,
           FBa2                     := #xTmp,
           Out                      := Q    171.2);

NETWORK
TITLE =A11_GOA_1102  Mixer A11 KEINE ANSTEUERUNG!!!
// Act 023
// Box           : FM-A11
// Output address: Q171.4
      CALL FC    70 (
           UnitNo                   := #UnitNo,
           ActRec                   := DB5110.A11_GOA_1102,
           Typ                      := 0,
           FBa                      := #xTmp,
           FBa2                     := #xTmp,
           Out                      := Q    171.4);

NETWORK
TITLE =A11_GOA_1103  Mixer A11 KEINE ANSTEUERUNG!!!
// Act 024
// Box           : FM-A11
// Output address: Q171.5
      CALL FC    70 (
           UnitNo                   := #UnitNo,
           ActRec                   := DB5110.A11_GOA_1103,
           Typ                      := 0,
           FBa                      := #xTmp,
           FBa2                     := #xTmp,
           Out                      := Q    171.5);

NETWORK
TITLE =A11_Schwenkbogen  "1"=CIP  "0"=Produktion
// Act 028
// Box           : Sirup
// Output address: DB_SEND_DOEHLER.Anlage11.Schwenkbogen
      CALL FC    70 (
           UnitNo                   := #UnitNo,
           ActRec                   := DB5110.A11_Schwenkbogen,
           Typ                      := 0,
           FBa                      := #xTmp,
           FBa2                     := #xTmp,
           Out                      := DB404.DBX   61.0);

NETWORK
TITLE =M11_MOLCH_ENDPOSITION  Mixer A11 Molch am Mixer in Endposition
// Act 034
// Box           : FM-A11
// Output address: Q171.7
      CALL FC    70 (
           UnitNo                   := #UnitNo,
           ActRec                   := DB5110.M11_MOLCH_ENDPOSITION,
           Typ                      := 0,
           FBa                      := #xTmp,
           FBa2                     := #xTmp,
           Out                      := #xTmp);//"M11_MOLCH_ENDPOSITIONO"

NETWORK
TITLE =A11_Molch_Sirup  "1"=Molch ist im Sirupraum
// Act 046
// Box           : Sirup
// Output address: DB_SEND_DOEHLER.Anlage11.Molch_Sirup
      CALL FC    70 (
           UnitNo                   := #UnitNo,
           ActRec                   := DB5110.A11_Molch_Sirup,
           Typ                      := 0,
           FBa                      := #xTmp,
           FBa2                     := #xTmp,
           Out                      := DB404.DBX   60.0);

NETWORK
TITLE =A11_Molch_Anlage  "1"=Molch ist an der Anlage
// Act 047
// Box           : Sirup
// Output address: DB_SEND_DOEHLER.Anlage11.Molch_Anlage
      CALL FC    70 (
           UnitNo                   := #UnitNo,
           ActRec                   := DB5110.A11_Molch_Anlage,
           Typ                      := 0,
           FBa                      := #xTmp,
           FBa2                     := #xTmp,
           Out                      := DB404.DBX   60.1);

NETWORK
TITLE =A11_Molch_PRO  "1"=Molch ist bereit für Produktion
// Act 048
// Box           : Sirup
// Output address: DB_SEND_DOEHLER.Anlage11.Molch_PRO
      CALL FC    70 (
           UnitNo                   := #UnitNo,
           ActRec                   := DB5110.A11_Molch_PRO,
           Typ                      := 0,
           FBa                      := #xTmp,
           FBa2                     := #xTmp,
           Out                      := DB404.DBX   60.2);

NETWORK
TITLE =A11_Molch_CIP  "1"=Molch ist bereit für CIP
// Act 049
// Box           : Sirup
// Output address: DB_SEND_DOEHLER.Anlage11.Molch_CIP
      CALL FC    70 (
           UnitNo                   := #UnitNo,
           ActRec                   := DB5110.A11_Molch_CIP,
           Typ                      := 0,
           FBa                      := #xTmp,
           FBa2                     := #xTmp,
           Out                      := DB404.DBX   60.3);

NETWORK
TITLE =A11_Sirupanforderung
// Act 050
// Box           : Sirup
// Output address: DB_SEND_DOEHLER.Anlage11.Sirupanforderung
      CALL FC    70 (
           UnitNo                   := #UnitNo,
           ActRec                   := DB5110.A11_Sirupanforderung,
           Typ                      := 0,
           FBa                      := #xTmp,
           FBa2                     := #xTmp,
           Out                      := DB404.DBX   60.4);

END_FUNCTION_BLOCK

FUNCTION_BLOCK FB 4111
TITLE =U111: Transfer Plant 11
FAMILY : BOTEC_F1
NAME : UniE
VERSION : 1.2


VAR_TEMP
  CIP : BOOL ;	//CIP active
  UNIM : BOOL ;	//Unit Not In Maintenance
  GenRel : BOOL ;	//general OK (emergency and maintenance OK)
  EStopOK : BOOL ;	//emergency OK
  UnitNo : INT ;	//unit number
  xTmp : BOOL ;	//Temporary Bool
  iTmp : INT ;	//Temporary INT
  rTmp : REAL ;	//Temporary REAL
  dTmp : DINT ;	//Temporary DINT (free for general use)
  RetValInt : INT ;	//return value
END_VAR
BEGIN
NETWORK
TITLE =General

      SET   ;
// Simulation ---------------------------------------------------------------
      A     DB4111.DBX 1357.7;
      CC    FB  4119; // "U111Sim"
      A     DB4111.DBX   17.3;
      =     DB4111.DBX 1357.7; //Help bit for simulation

// get unit number ----------------------------------------------------------
      L     DB4110.DBW    0;
      T     #UnitNo;

// communication ------------------------------------------------------------
      UC    FB  4115; // U111Com

NETWORK
TITLE =Sequence organisation

      CLR   ;
      =     M    122.2;

// sequencer ----------------------------------------------------------------
      A     DB4113.DBX   43.1;
      S     DB4113.DBX   97.3;

      CALL FC    40 (
           UnitNo                   := #UnitNo);

END_FUNCTION_BLOCK

FUNCTION_BLOCK FB 4120
TITLE =U112: Sirup Anlage 12
FAMILY : BOTEC_F1
NAME : U112A
VERSION : 2.1


VAR_TEMP
  EStopOK : BOOL ;	//auxiliary flag
  CIP : BOOL ;	//CIP Program Selected
  xTmp : BOOL ;	//Temporary Bool(free for general use)
  DummyBool : BOOL ;	//Temporary Bool(free for general use)
  UnitNo : INT ;	//unit number
  UnitFB : INT ;	//unit expansion FB number
  rTmp : REAL ;	//Temporary REAL (free for general use)
  iTmp : INT ;	//Temporary INT (free for general use)
  DummyInt : INT ;	//Temporary INT (free for general use)
  dTmp : DINT ;	//Temporary DINT (free for general use)
END_VAR
BEGIN
NETWORK
TITLE =general

      CLR   ;
      =     #xTmp;
      =     #EStopOK;

      L     DB4120.DBW    0;
      T     #UnitNo;
      L     DB4120.DBW    2;
      T     #UnitFB;

NETWORK
TITLE =Universal value

      NOP   0;
// unv001 UnV 001 Process Status
      CALL FC    27 (
           UnitNo                   := #UnitNo,
           UnVRec                   := DB5125.unv001,
           ValExt                   := DB5125.DBD  234);

// unv002 UnV 002 Universal Value 02
      CALL FC    27 (
           UnitNo                   := #UnitNo,
           UnVRec                   := DB5125.unv002,
           ValExt                   := DB5125.DBD  362);

// unv003 UnV 003 Universal Value 03
      CALL FC    27 (
           UnitNo                   := #UnitNo,
           UnVRec                   := DB5125.unv003,
           ValExt                   := DB5125.DBD  490);

// unv004 UnV 004 Universal Value 04
      CALL FC    27 (
           UnitNo                   := #UnitNo,
           UnVRec                   := DB5125.unv004,
           ValExt                   := DB5125.DBD  618);

NETWORK
TITLE =special inputs

      NOP   0;
// GOA_SA12_31_oben SpI 004
      CALL FC    14 (
           UnitNo                   := #UnitNo,
           SpIRec                   := DB5121.GOA_SA12_31_oben,
           SpIBit                   := I    267.6);

// GOA_SA12_41_unten SpI 005
      CALL FC    14 (
           UnitNo                   := #UnitNo,
           SpIRec                   := DB5121.GOA_SA12_41_unten,
           SpIBit                   := I    267.7);

// GOA_SA12_1 SpI 006
      CALL FC    14 (
           UnitNo                   := #UnitNo,
           SpIRec                   := DB5121.GOA_SA12_1,
           SpIBit                   := I    267.4);

// GOA_SA12_2 SpI 007
      CALL FC    14 (
           UnitNo                   := #UnitNo,
           SpIRec                   := DB5121.GOA_SA12_2,
           SpIBit                   := I    267.5);

// SK_A12_Molch_Abbruch_DT SpI 008 MOLCH A12 Drucktaste Abbruch Sirupraum
      CALL FC    14 (
           UnitNo                   := #UnitNo,
           SpIRec                   := DB5121.SK_A12_Molch_Abbruch_DT,
           SpIBit                   := I    264.0);

// SK_A12_START_Molch_LDT SpI 009 MOLCH A12 L-Drucktaste Start Sirupraum
      CALL FC    14 (
           UnitNo                   := #UnitNo,
           SpIRec                   := DB5121.SK_A12_START_Molch_LDT,
           SpIBit                   := I    264.3);

// A12_K1_Handklappe SpI 010 Handklappe Sirupraum Molch Anlage 12
      CALL FC    14 (
           UnitNo                   := #UnitNo,
           SpIRec                   := DB5121.A12_K1_Handklappe,
           SpIBit                   := I    267.3);

// GOA_EA12_31_oben SpI 014
      CALL FC    14 (
           UnitNo                   := #UnitNo,
           SpIRec                   := DB5121.GOA_EA12_31_oben,
           SpIBit                   := I    262.5);

// GOA_EA12_32_unten SpI 015
      CALL FC    14 (
           UnitNo                   := #UnitNo,
           SpIRec                   := DB5121.GOA_EA12_32_unten,
           SpIBit                   := I    262.6);

// GOA_EA12_3 SpI 016
      CALL FC    14 (
           UnitNo                   := #UnitNo,
           SpIRec                   := DB5121.GOA_EA12_3,
           SpIBit                   := I    262.3);

// GOA_EA12_4 SpI 017
      CALL FC    14 (
           UnitNo                   := #UnitNo,
           SpIRec                   := DB5121.GOA_EA12_4,
           SpIBit                   := I    262.4);

// A12_SS_FRG_MOLCH SpI 018 Anlage 12 Schlüsselschalter Freigabe Molch
      CALL FC    14 (
           UnitNo                   := #UnitNo,
           SpIRec                   := DB5121.A12_SS_FRG_MOLCH,
           SpIBit                   := I    263.4);

// A12_Molch_LDT_Start SpI 019
      CALL FC    14 (
           UnitNo                   := #UnitNo,
           SpIRec                   := DB5121.A12_Molch_LDT_Start,
           SpIBit                   := I    262.7);

// A12_Molch_LDT_Stop SpI 020
      CALL FC    14 (
           UnitNo                   := #UnitNo,
           SpIRec                   := DB5121.A12_Molch_LDT_Stop,
           SpIBit                   := I    263.5);

// A12_K2_Handklappe SpI 021
      CALL FC    14 (
           UnitNo                   := #UnitNo,
           SpIRec                   := DB5121.A12_K2_Handklappe,
           SpIBit                   := I    263.2);

// GOA_1201 SpI 022
      CALL FC    14 (
           UnitNo                   := #UnitNo,
           SpIRec                   := DB5121.GOA_1201,
           SpIBit                   := I    262.0);

// GOA_1202 SpI 023
      CALL FC    14 (
           UnitNo                   := #UnitNo,
           SpIRec                   := DB5121.GOA_1202,
           SpIBit                   := I    262.1);

// GOA_1204 SpI 025 Schwenkbogen CIP 3
      CALL FC    14 (
           UnitNo                   := #UnitNo,
           SpIRec                   := DB5121.GOA_1204,
           SpIBit                   := I    263.3);

NETWORK
TITLE =messages

      NOP   0;
// msg001 Msg 001 Message 01
      CALL FC    16 (
           UnitNo                   := #UnitNo,
           MsgRec                   := DB5127.msg001,
           MsgBit                   := DB5127.DBX   82.7);

// msg002 Msg 002 Message 02
      CALL FC    16 (
           UnitNo                   := #UnitNo,
           MsgRec                   := DB5127.msg002,
           MsgBit                   := DB5127.DBX  142.7);

// msg003 Msg 003 Message 03
      CALL FC    16 (
           UnitNo                   := #UnitNo,
           MsgRec                   := DB5127.msg003,
           MsgBit                   := DB5127.DBX  202.7);

NETWORK
TITLE =unit supply

      UC    FB [#UnitFB];

NETWORK
TITLE =A12_MWV1  MOLCH A12 Ansteuerung MWV1
// Act 002
// Box           : VS-SRA
// Input address : I189.2
// Output address: Q189.2
      CALL FC    70 (
           UnitNo                   := #UnitNo,
           ActRec                   := DB5120.A12_MWV1,
           Typ                      := 1,
           FBa                      := #xTmp,
           FBa2                     := I    189.2,
           Out                      := Q    189.2);

NETWORK
TITLE =SA12_V2  MOLCH SA12 Ansteuerung V2
// Act 003
// Box           : VS-SRA
// Input address : I189.3
// Output address: Q189.3
      CALL FC    70 (
           UnitNo                   := #UnitNo,
           ActRec                   := DB5120.SA12_V2,
           Typ                      := 1,
           FBa                      := #xTmp,
           FBa2                     := I    189.3,
           Out                      := Q    189.3);

NETWORK
TITLE =SA12_V31  MOLCH SA12 Ansteuerung V31 (ohne RM)
// Act 004
// Box           : VS-SRA
// Output address: Q188.6
      CALL FC    70 (
           UnitNo                   := #UnitNo,
           ActRec                   := DB5120.SA12_V31,
           Typ                      := 0,
           FBa                      := #xTmp,
           FBa2                     := #xTmp,
           Out                      := Q    188.6);

NETWORK
TITLE =SA12_V32  MOLCH SA12 Ansteuerung V32 (ohne RM)
// Act 005
// Box           : VS-SRA
// Output address: Q188.7
      CALL FC    70 (
           UnitNo                   := #UnitNo,
           ActRec                   := DB5120.SA12_V32,
           Typ                      := 0,
           FBa                      := #xTmp,
           FBa2                     := #xTmp,
           Out                      := Q    188.7);

NETWORK
TITLE =SA12_V41  MOLCH SA12 Ansteuerung V41
// Act 006
// Box           : VS-SRA
// Input address : I189.0
// Output address: Q189.0
      CALL FC    70 (
           UnitNo                   := #UnitNo,
           ActRec                   := DB5120.SA12_V41,
           Typ                      := 1,
           FBa                      := #xTmp,
           FBa2                     := I    189.0,
           Out                      := Q    189.0);

NETWORK
TITLE =SA12_V42  MOLCH SA12 Ansteuerung V42
// Act 007
// Box           : VS-SRA
// Input address : I189.1
// Output address: Q189.1
      CALL FC    70 (
           UnitNo                   := #UnitNo,
           ActRec                   := DB5120.SA12_V42,
           Typ                      := 1,
           FBa                      := #xTmp,
           FBa2                     := I    189.1,
           Out                      := Q    189.1);

NETWORK
TITLE =SK_A12_Abbruch_L  Anlage 12 Lampe Abbruch IM SIRUPRAUM
// Act 008
// Box           : AB1SK
// Output address: Q264.2
      CALL FC    70 (
           UnitNo                   := #UnitNo,
           ActRec                   := DB5120.SK_A12_Abbruch_L,
           Typ                      := 0,
           FBa                      := #xTmp,
           FBa2                     := #xTmp,
           Out                      := Q    264.2);

NETWORK
TITLE =SK_A12_START_Molch_L  Anlage 12 Lampe Start Molch IM SIRUPRAUM
// Act 009
// Box           : AB1SK
// Output address: Q264.3
      CALL FC    70 (
           UnitNo                   := #UnitNo,
           ActRec                   := DB5120.SK_A12_START_Molch_L,
           Typ                      := 0,
           FBa                      := #xTmp,
           FBa2                     := #xTmp,
           Out                      := Q    264.3);

NETWORK
TITLE =A12_MOLCH_A12_L  Anlage 12 Lampe Molch an A12 IM SIRUPRAUM
// Act 010
// Box           : AB1SK
// Output address: Q264.0
      CALL FC    70 (
           UnitNo                   := #UnitNo,
           ActRec                   := DB5120.A12_MOLCH_A12_L,
           Typ                      := 0,
           FBa                      := #xTmp,
           FBa2                     := #xTmp,
           Out                      := Q    264.0);

NETWORK
TITLE =SK_A12_MOLCH_IN_SK_L  Anlage 12 Lampe Molch im SK IM SIRUPRAUM
// Act 011
// Box           : AB1SK
// Output address: Q264.1
      CALL FC    70 (
           UnitNo                   := #UnitNo,
           ActRec                   := DB5120.SK_A12_MOLCH_IN_SK_L,
           Typ                      := 0,
           FBa                      := #xTmp,
           FBa2                     := #xTmp,
           Out                      := Q    264.1);

NETWORK
TITLE =EA12_V1  A12 V1
// Act 012
// Box           : VSA12
// Input address : I260.4
// Output address: Q260.4
      CALL FC    70 (
           UnitNo                   := #UnitNo,
           ActRec                   := DB5120.EA12_V1,
           Typ                      := 1,
           FBa                      := #xTmp,
           FBa2                     := I    260.4,
           Out                      := Q    260.4);

NETWORK
TITLE =EA12_V2  A12 V2
// Act 013
// Box           : VSA12
// Input address : I260.5
// Output address: Q260.5
      CALL FC    70 (
           UnitNo                   := #UnitNo,
           ActRec                   := DB5120.EA12_V2,
           Typ                      := 1,
           FBa                      := #xTmp,
           FBa2                     := I    260.5,
           Out                      := Q    260.5);

NETWORK
TITLE =EA12_V31  A12 V31 ohne RM
// Act 014
// Box           : VSA12
// Input address : I260.0
// Output address: Q260.0
      CALL FC    70 (
           UnitNo                   := #UnitNo,
           ActRec                   := DB5120.EA12_V31,
           Typ                      := 0,
           FBa                      := #xTmp,
           FBa2                     := I    260.0,
           Out                      := Q    260.0);

NETWORK
TITLE =EA12_V32  A12 V31 ohne RM
// Act 015
// Box           : VSA12
// Input address : I260.1
// Output address: Q260.1
      CALL FC    70 (
           UnitNo                   := #UnitNo,
           ActRec                   := DB5120.EA12_V32,
           Typ                      := 0,
           FBa                      := #xTmp,
           FBa2                     := I    260.1,
           Out                      := Q    260.1);

NETWORK
TITLE =EA12_V41  A12 V41
// Act 016
// Box           : VSA12
// Input address : I260.2
// Output address: Q260.2
      CALL FC    70 (
           UnitNo                   := #UnitNo,
           ActRec                   := DB5120.EA12_V41,
           Typ                      := 1,
           FBa                      := #xTmp,
           FBa2                     := I    260.2,
           Out                      := Q    260.2);

NETWORK
TITLE =EA12_V42  A12 V42
// Act 017
// Box           : VSA12
// Input address : I260.3
// Output address: Q260.3
      CALL FC    70 (
           UnitNo                   := #UnitNo,
           ActRec                   := DB5120.EA12_V42,
           Typ                      := 1,
           FBa                      := #xTmp,
           FBa2                     := I    260.3,
           Out                      := Q    260.3);

NETWORK
TITLE =EA12_MOLCH_LDT_Start  Leuchtdrucktaster START Molch Anlage 12
// Act 019
// Box           : VSA12
// Output address: Q262.7
      CALL FC    70 (
           UnitNo                   := #UnitNo,
           ActRec                   := DB5120.EA12_MOLCH_LDT_Start,
           Typ                      := 0,
           FBa                      := #xTmp,
           FBa2                     := #xTmp,
           Out                      := Q    262.7);

NETWORK
TITLE =Molch ist unterwegs (Mixer)


      CALL FC    70 (
           UnitNo                   := #UnitNo,
           ActRec                   := DB5120.Act20,
           Typ                      := 0,
           FBa                      := #xTmp,
           FBa2                     := #xTmp,
           Out                      := Q    271.3);

NETWORK
TITLE =Molch in Endposition (Mixer)


      CALL FC    70 (
           UnitNo                   := #UnitNo,
           ActRec                   := DB5120.Act21,
           Typ                      := 0,
           FBa                      := #xTmp,
           FBa2                     := #xTmp,
           Out                      := Q    271.7);

NETWORK
TITLE =A12_Schwenkbogen  "1"=CIP  "0"=Produktion
// Act 028
// Box           : Sirup
// Output address: DB_SEND_DOEHLER.Anlage12.Schwenkbogen
      CALL FC    70 (
           UnitNo                   := #UnitNo,
           ActRec                   := DB5120.A12_Schwenkbogen,
           Typ                      := 0,
           FBa                      := #xTmp,
           FBa2                     := #xTmp,
           Out                      := DB404.DBX   63.0);

NETWORK
TITLE =A12_Molch_Sirup  "1"=Molch ist im Sirupraum
// Act 046
// Box           : Sirup
// Output address: DB_SEND_DOEHLER.Anlage12.Molch_Sirup
      CALL FC    70 (
           UnitNo                   := #UnitNo,
           ActRec                   := DB5120.A12_Molch_Sirup,
           Typ                      := 0,
           FBa                      := #xTmp,
           FBa2                     := #xTmp,
           Out                      := DB404.DBX   62.0);

NETWORK
TITLE =A12_Molch_Anlage  "1"=Molch ist an der Anlage
// Act 047
// Box           : Sirup
// Output address: DB_SEND_DOEHLER.Anlage12.Molch_Anlage
      CALL FC    70 (
           UnitNo                   := #UnitNo,
           ActRec                   := DB5120.A12_Molch_Anlage,
           Typ                      := 0,
           FBa                      := #xTmp,
           FBa2                     := #xTmp,
           Out                      := DB404.DBX   62.1);

NETWORK
TITLE =A12_Molch_PRO  "1"=Molch ist bereit für Produktion
// Act 048
// Box           : Sirup
// Output address: DB_SEND_DOEHLER.Anlage12.Molch_PRO
      CALL FC    70 (
           UnitNo                   := #UnitNo,
           ActRec                   := DB5120.A12_Molch_PRO,
           Typ                      := 0,
           FBa                      := #xTmp,
           FBa2                     := #xTmp,
           Out                      := DB404.DBX   62.2);

NETWORK
TITLE =A12_Molch_CIP  "1"=Molch ist bereit für CIP
// Act 049
// Box           : Sirup
// Output address: DB_SEND_DOEHLER.Anlage12.Molch_CIP
      CALL FC    70 (
           UnitNo                   := #UnitNo,
           ActRec                   := DB5120.A12_Molch_CIP,
           Typ                      := 0,
           FBa                      := #xTmp,
           FBa2                     := #xTmp,
           Out                      := DB404.DBX   62.3);

NETWORK
TITLE =A12_Sirupanforderung
// Act 050
// Box           : Sirup
// Output address: DB_SEND_DOEHLER.Anlage12.Sirupanforderung
      CALL FC    70 (
           UnitNo                   := #UnitNo,
           ActRec                   := DB5120.A12_Sirupanforderung,
           Typ                      := 0,
           FBa                      := #xTmp,
           FBa2                     := #xTmp,
           Out                      := DB404.DBX   62.4);

END_FUNCTION_BLOCK

FUNCTION_BLOCK FB 4121
TITLE =U112: Transfer Plant 12
FAMILY : BOTEC_F1
NAME : UniE
VERSION : 1.2


VAR_TEMP
  CIP : BOOL ;	//CIP active
  UNIM : BOOL ;	//Unit Not In Maintenance
  GenRel : BOOL ;	//general OK (emergency and maintenance OK)
  EStopOK : BOOL ;	//emergency OK
  UnitNo : INT ;	//unit number
  xTmp : BOOL ;	//Temporary Bool
  iTmp : INT ;	//Temporary INT
  rTmp : REAL ;	//Temporary REAL
  dTmp : DINT ;	//Temporary DINT (free for general use)
  RetValInt : INT ;	//return value
END_VAR
BEGIN
NETWORK
TITLE =General

      SET   ;
// Simulation ---------------------------------------------------------------
      A     DB4121.DBX 1357.7;
      CC    FB  4129; // "U112Sim"
      A     DB4121.DBX   17.3;
      =     DB4121.DBX 1357.7; //Help bit for simulation

// get unit number ----------------------------------------------------------
      L     DB4120.DBW    0;
      T     #UnitNo;

// communication ------------------------------------------------------------
      UC    FB  4125; // U112Com

NETWORK
TITLE =Sequence organisation

      CLR   ;
      =     M    122.2;


// sequencer ----------------------------------------------------------------
      A     DB4123.DBX   43.1;
      S     DB4123.DBX   97.3;

      CALL FC    40 (
           UnitNo                   := #UnitNo);

END_FUNCTION_BLOCK

FUNCTION_BLOCK FB 4140
TITLE =U114: Sirup Anlage 14
FAMILY : BOTEC_F1
NAME : U114A
VERSION : 2.1


VAR_TEMP
  EStopOK : BOOL ;	//auxiliary flag
  CIP : BOOL ;	//CIP Program Selected
  xTmp : BOOL ;	//Temporary Bool(free for general use)
  DummyBool : BOOL ;	//Temporary Bool(free for general use)
  UnitNo : INT ;	//unit number
  UnitFB : INT ;	//unit expansion FB number
  rTmp : REAL ;	//Temporary REAL (free for general use)
  iTmp : INT ;	//Temporary INT (free for general use)
  DummyInt : INT ;	//Temporary INT (free for general use)
  dTmp : DINT ;	//Temporary DINT (free for general use)
END_VAR
BEGIN
NETWORK
TITLE =general

      CLR   ;
      =     #xTmp;
      =     #EStopOK;

      L     DB4140.DBW    0;
      T     #UnitNo;
      L     DB4140.DBW    2;
      T     #UnitFB;

NETWORK
TITLE =Universal value

      NOP   0;
// unv001 UnV 001 Process Status
      CALL FC    27 (
           UnitNo                   := #UnitNo,
           UnVRec                   := DB5145.unv001,
           ValExt                   := DB5145.DBD  234);

// unv002 UnV 002 Universal Value 02
      CALL FC    27 (
           UnitNo                   := #UnitNo,
           UnVRec                   := DB5145.unv002,
           ValExt                   := DB5145.DBD  362);

// unv003 UnV 003 Universal Value 03
      CALL FC    27 (
           UnitNo                   := #UnitNo,
           UnVRec                   := DB5145.unv003,
           ValExt                   := DB5145.DBD  490);

// unv004 UnV 004 Universal Value 04
      CALL FC    27 (
           UnitNo                   := #UnitNo,
           UnVRec                   := DB5145.unv004,
           ValExt                   := DB5145.DBD  618);

NETWORK
TITLE =special inputs

      NOP   0;
// GOA_SA14_31_oben SpI 004 GOA_SA14_31_oben
      CALL FC    14 (
           UnitNo                   := #UnitNo,
           SpIRec                   := DB5141.GOA_SA14_31_oben,
           SpIBit                   := I    266.4);

// GOA_SA14_32_unten SpI 005 GOA_SA14_32_unten
      CALL FC    14 (
           UnitNo                   := #UnitNo,
           SpIRec                   := DB5141.GOA_SA14_32_unten,
           SpIBit                   := I    266.5);

// GOA_SA14_2 SpI 006 GOA_SA14_2
      CALL FC    14 (
           UnitNo                   := #UnitNo,
           SpIRec                   := DB5141.GOA_SA14_2,
           SpIBit                   := I    266.3);

// GOA_SA14_1 SpI 007 GOA_SA14_1
      CALL FC    14 (
           UnitNo                   := #UnitNo,
           SpIRec                   := DB5141.GOA_SA14_1,
           SpIBit                   := I    266.2);

// SK_A14_Molch_Abbruch_DT SpI 008 MOLCH A14 Drucktaste Abbruch Sirupraum
      CALL FC    14 (
           UnitNo                   := #UnitNo,
           SpIRec                   := DB5141.SK_A14_Molch_Abbruch_DT,
           SpIBit                   := I    265.2);

// SK_A14_START_Molch_LDT SpI 009 MOLCH A14 L-Drucktaste Start Sirupraum
      CALL FC    14 (
           UnitNo                   := #UnitNo,
           SpIRec                   := DB5141.SK_A14_START_Molch_LDT,
           SpIBit                   := I    265.5);

// GOA_EA14_31_OBEN SpI 014
      CALL FC    14 (
           UnitNo                   := #UnitNo,
           SpIRec                   := DB5141.GOA_EA14_31_OBEN,
           SpIBit                   := I     98.5);

// GOA_EA14_32_UNTEN SpI 015
      CALL FC    14 (
           UnitNo                   := #UnitNo,
           SpIRec                   := DB5141.GOA_EA14_32_UNTEN,
           SpIBit                   := I     98.6);

// GOA_EA14_3 SpI 016
      CALL FC    14 (
           UnitNo                   := #UnitNo,
           SpIRec                   := DB5141.GOA_EA14_3,
           SpIBit                   := I     98.3);

// GOA_EA14_4 SpI 017
      CALL FC    14 (
           UnitNo                   := #UnitNo,
           SpIRec                   := DB5141.GOA_EA14_4,
           SpIBit                   := I     98.4);

// A14_FREIGABE_MOLCH_SS SpI 018
      CALL FC    14 (
           UnitNo                   := #UnitNo,
           SpIRec                   := DB5141.A14_FREIGABE_MOLCH_SS,
           SpIBit                   := I     99.4);

// A14_MOLCH_START_LDT SpI 019
      CALL FC    14 (
           UnitNo                   := #UnitNo,
           SpIRec                   := DB5141.A14_MOLCH_START_LDT,
           SpIBit                   := I     98.7);

// A14_MOLCH_STOP_DT SpI 020
      CALL FC    14 (
           UnitNo                   := #UnitNo,
           SpIRec                   := DB5141.A14_MOLCH_STOP_DT,
           SpIBit                   := I     99.5);

// GOA_1405 SpI 021
      CALL FC    14 (
           UnitNo                   := #UnitNo,
           SpIRec                   := DB5141.GOA_1405,
           SpIBit                   := I     99.3);

// GOA_1401 SpI 022
      CALL FC    14 (
           UnitNo                   := #UnitNo,
           SpIRec                   := DB5141.GOA_1401,
           SpIBit                   := I     98.0);

// GOA_1402 SpI 023
      CALL FC    14 (
           UnitNo                   := #UnitNo,
           SpIRec                   := DB5141.GOA_1402,
           SpIBit                   := I     98.1);

// GOA_1404 SpI 025
      CALL FC    14 (
           UnitNo                   := #UnitNo,
           SpIRec                   := DB5141.GOA_1404,
           SpIBit                   := I     99.2);

NETWORK
TITLE =messages

      NOP   0;
// msg001 Msg 001 Message 01
      CALL FC    16 (
           UnitNo                   := #UnitNo,
           MsgRec                   := DB5147.msg001,
           MsgBit                   := DB5147.DBX   82.7);

// msg002 Msg 002 Message 02
      CALL FC    16 (
           UnitNo                   := #UnitNo,
           MsgRec                   := DB5147.msg002,
           MsgBit                   := DB5147.DBX  142.7);

// msg003 Msg 003 Message 03
      CALL FC    16 (
           UnitNo                   := #UnitNo,
           MsgRec                   := DB5147.msg003,
           MsgBit                   := DB5147.DBX  202.7);

NETWORK
TITLE =unit supply

      UC    FB [#UnitFB];

NETWORK
TITLE =A14_MWV1  MOLCH A14 Ansteuerung MWV1
// Act 002
// Box           : VS-SRA
// Input address : I190.6
// Output address: Q190.6
      CALL FC    70 (
           UnitNo                   := #UnitNo,
           ActRec                   := DB5140.A14_MWV1,
           Typ                      := 1,
           FBa                      := #xTmp,
           FBa2                     := I    190.6,
           Out                      := Q    190.6);

NETWORK
TITLE =SA14_V2  MOLCH SA14 Ansteuerung V2
// Act 003
// Box           : VS-SRA
// Input address : I190.7
// Output address: Q190.7
      CALL FC    70 (
           UnitNo                   := #UnitNo,
           ActRec                   := DB5140.SA14_V2,
           Typ                      := 1,
           FBa                      := #xTmp,
           FBa2                     := I    190.7,
           Out                      := Q    190.7);

NETWORK
TITLE =SA14_V31  MOLCH SA14 Ansteuerung V31 (ohne RM)
// Act 004
// Box           : VS-SRA
// Output address: Q190.2
      CALL FC    70 (
           UnitNo                   := #UnitNo,
           ActRec                   := DB5140.SA14_V31,
           Typ                      := 0,
           FBa                      := #xTmp,
           FBa2                     := #xTmp,
           Out                      := Q    190.2);

NETWORK
TITLE =SA14_V32  MOLCH SA14 Ansteuerung V32 (ohne RM)
// Act 005
// Box           : VS-SRA
// Output address: Q190.3
      CALL FC    70 (
           UnitNo                   := #UnitNo,
           ActRec                   := DB5140.SA14_V32,
           Typ                      := 0,
           FBa                      := #xTmp,
           FBa2                     := #xTmp,
           Out                      := Q    190.3);

NETWORK
TITLE =SA14_V41  MOLCH SA14 Ansteuerung V41
// Act 006
// Box           : VS-SRA
// Input address : I190.4
// Output address: Q190.4
      CALL FC    70 (
           UnitNo                   := #UnitNo,
           ActRec                   := DB5140.SA14_V41,
           Typ                      := 1,
           FBa                      := #xTmp,
           FBa2                     := I    190.4,
           Out                      := Q    190.4);

NETWORK
TITLE =SA14_V42  MOLCH SA14 Ansteuerung V42
// Act 007
// Box           : VS-SRA
// Input address : I190.5
// Output address: Q190.5
      CALL FC    70 (
           UnitNo                   := #UnitNo,
           ActRec                   := DB5140.SA14_V42,
           Typ                      := 1,
           FBa                      := #xTmp,
           FBa2                     := I    190.5,
           Out                      := Q    190.5);

NETWORK
TITLE =SK_A14_Abbruch_Stoerung  Anlage 14 Lampe Abbruch IM SIRUPRAUM
// Act 008
// Box           : AB1SK
// Output address: Q265.4
      CALL FC    70 (
           UnitNo                   := #UnitNo,
           ActRec                   := DB5140.SK_A14_Abbruch_Stoerung,
           Typ                      := 0,
           FBa                      := #xTmp,
           FBa2                     := #xTmp,
           Out                      := Q    265.4);

NETWORK
TITLE =SK_A14_Molch_Start_LDT  Anlage 14 Lampe Start Molch IM SIRUPRAUM
// Act 009
// Box           : AB1SK
// Output address: Q265.5
      CALL FC    70 (
           UnitNo                   := #UnitNo,
           ActRec                   := DB5140.SK_A14_Molch_Start_LDT,
           Typ                      := 0,
           FBa                      := #xTmp,
           FBa2                     := #xTmp,
           Out                      := Q    265.5);

NETWORK
TITLE =SK_A14_Molch_bei_A14  Anlage 14 Lampe Molch an A11 IM SIRUPRAUM
// Act 010
// Box           : AB1SK
// Output address: Q265.2
      CALL FC    70 (
           UnitNo                   := #UnitNo,
           ActRec                   := DB5140.SK_A14_Molch_bei_A14,
           Typ                      := 0,
           FBa                      := #xTmp,
           FBa2                     := #xTmp,
           Out                      := Q    265.2);

NETWORK
TITLE =SK_A14_Molch_in_SK  Anlage 14 Lampe Molch im SK IM SIRUPRAUM
// Act 011
// Box           : AB1SK
// Output address: Q265.3
      CALL FC    70 (
           UnitNo                   := #UnitNo,
           ActRec                   := DB5140.SK_A14_Molch_in_SK,
           Typ                      := 0,
           FBa                      := #xTmp,
           FBa2                     := #xTmp,
           Out                      := Q    265.3);

NETWORK
TITLE =EA14_V1
// Act 012
// Box           : VSA14
// Input address : I96.4
// Output address: Q96.4
      CALL FC    70 (
           UnitNo                   := #UnitNo,
           ActRec                   := DB5140.EA14_V1,
           Typ                      := 1,
           FBa                      := #xTmp,
           FBa2                     := I     96.4,
           Out                      := Q     96.4);

NETWORK
TITLE =EA14_V2
// Act 013
// Box           : VSA14
// Input address : I96.5
// Output address: Q96.5
      CALL FC    70 (
           UnitNo                   := #UnitNo,
           ActRec                   := DB5140.EA14_V2,
           Typ                      := 1,
           FBa                      := #xTmp,
           FBa2                     := I     96.5,
           Out                      := Q     96.5);

NETWORK
TITLE =EA14_V31  EA14 V31 (ohne Rückmeldung)
// Act 014
// Box           : VSA14
// Output address: Q96.0
      CALL FC    70 (
           UnitNo                   := #UnitNo,
           ActRec                   := DB5140.EA14_V31,
           Typ                      := 0,
           FBa                      := #xTmp,
           FBa2                     := #xTmp,
           Out                      := Q     96.0);

NETWORK
TITLE =EA14_V32  EA14 V32 (ohne Rückmeldung)
// Act 015
// Box           : VSA14
// Output address: Q96.1
      CALL FC    70 (
           UnitNo                   := #UnitNo,
           ActRec                   := DB5140.EA14_V32,
           Typ                      := 0,
           FBa                      := #xTmp,
           FBa2                     := #xTmp,
           Out                      := Q     96.1);

